{attribute 'no_explicit_call' := 'do not call this function block directly'} 
FUNCTION_BLOCK ABSTRACT GenericList EXTENDS Object IMPLEMENTS IList
VAR_INPUT
	DefaultAllocationElemetsCount : BYTE := 10;	
END_VAR
VAR_OUTPUT
	StoredTypeCategory : TYPE_CATEGORY;
END_VAR
VAR
	_Array : POINTER TO GENERIC_VALUE;
	_ArrayLength : DINT;
	_ValueCount : DINT;
END_VAR

METHOD AllocateMemory
VAR_INPUT
	elementsCount : DINT;
END_VAR
VAR	
	newMemory : POINTER TO GENERIC_VALUE;
END_VAR
newMemory := __NEW(BYTE, TO_UDINT(SIZEOF(GENERIC_VALUE) * (_ArrayLength + elementsCount)));

IF _ValueCount > 0 THEN
	Tc2_System.MEMCPY(newMemory, _Array, TO_UDINT(SIZEOF(GENERIC_VALUE) * _ValueCount));
END_IF
 
IF _Array <> 0 THEN
	__DELETE(_Array);
END_IF

_ArrayLength := _ArrayLength + elementsCount;

_Array := newMemory;
END_METHOD

METHOD Append : DINT
VAR_INPUT
	value : ANY;
	isObject : BOOL := FALSE;
END_VAR
VAR
	genericValue : GENERIC_VALUE;
END_VAR
genericValue.FromAnyType(value, isObject, StoredTypeCategory = TYPE_CATEGORY.VALUE_TYPE);

Append := AppendGenericValue(genericValue);
END_METHOD

METHOD PROTECTED AppendGenericValue : DINT
VAR_IN_OUT CONSTANT
	value : GENERIC_VALUE;
END_VAR
AppendGenericValue := _ValueCount;

InsertGenericValue(value, AppendGenericValue);
END_METHOD

METHOD Clear
VAR
	i : DINT;
END_VAR
IF _ValueCount > 0 AND_THEN StoredTypeCategory = TYPE_CATEGORY.VALUE_TYPE THEN
	FOR i := 0 TO _ValueCount - 1 DO
		_Array[i].ReleaseOwnedMemory();						
	END_FOR	
END_IF

_ValueCount := 0;
_ArrayLength := 0;

IF _Array <> 0 THEN
	__DELETE(_Array);	
END_IF
END_METHOD

{attribute 'OPC.UA.DA.Property' := '1'}
{attribute 'monitoring' := 'call'}
PROPERTY Count : DINT
GET
Count := _ValueCount;
END_GET
END_PROPERTY

METHOD CreateEnumerator : IEnumerator
VAR
	listEnumerator : POINTER TO ListEnumerator;
END_VAR
listEnumerator := __NEW(ListEnumerator(list := THIS^));

CreateEnumerator := listEnumerator^;
END_METHOD

METHOD FB_exit : BOOL
VAR_INPUT
	bInCopyCode : BOOL; // if TRUE, the exit method is called for exiting an instance that is copied afterwards (online change).
END_VAR
Clear();
END_METHOD

METHOD FindSingle : BOOL
VAR_INPUT
	predicate : IPredicate;
	skip : UDINT := 0;
	searchDirection : SEARCH_DIRECTION := SEARCH_DIRECTION.FROM_BEGINNING;
END_VAR
VAR_OUTPUT
	value : GENERIC_VALUE;
	index : DINT;
END_VAR
VAR
	startSearchIndex : DINT;
	maxSearchIndex : DINT;
	indexStep : DINT;
	i : DINT;
	skiped : UDINT := 0;
END_VAR
index := 0;
	
IF TO_DINT(skip) >= _ValueCount OR_ELSE predicate = 0 THEN
	RETURN;
END_IF

startSearchIndex := SEL(searchDirection = SEARCH_DIRECTION.FROM_BEGINNING, _ValueCount - 1, 0);
maxSearchIndex := SEL(searchDirection = SEARCH_DIRECTION.FROM_BEGINNING, 0, _ValueCount - 1);
indexStep := SEL(searchDirection = SEARCH_DIRECTION.FROM_BEGINNING, -1, 1);

FOR i := startSearchIndex TO maxSearchIndex BY indexStep DO
	IF predicate.Compare(_Array[i].AsAnyType()) THEN
		IF skip = skiped THEN
			value := _Array[i];
			index := i;
			FindSingle := TRUE;
			RETURN;
		ELSE
			skiped := skiped + 1;
		END_IF
	END_IF
END_FOR
END_METHOD

METHOD Get : REFERENCE TO GENERIC_VALUE
VAR_INPUT
	index : DINT;
END_VAR
VAR
	argumentOutOfRangeException : ArgumentOutOfRangeException;
END_VAR
IF index < 0 OR index >= _ValueCount THEN
	argumentOutOfRangeException.Throw(CurrentNamespace.Name, ClassName, __POUNAME(), __POSITION(), 'index', index);
END_IF

Get REF= _Array[index];
END_METHOD

METHOD Insert
VAR_INPUT
	value : ANY;
	index : DINT;
	isObject : BOOL := FALSE;
END_VAR
VAR
	genericValue : GENERIC_VALUE;
END_VAR
genericValue.FromAnyType(value, isObject, StoredTypeCategory = TYPE_CATEGORY.VALUE_TYPE);

InsertGenericValue(genericValue, index);
END_METHOD

METHOD PROTECTED InsertGenericValue
VAR_IN_OUT CONSTANT
	value : GENERIC_VALUE;	
END_VAR
VAR_INPUT
	index : DINT;
END_VAR
VAR
	argumentOutOfRangeException : ArgumentOutOfRangeException;
	i : DINT;
END_VAR
IF index < 0 OR index > _ValueCount THEN
	argumentOutOfRangeException.Throw(CurrentNamespace.Name, ClassName, __POUNAME(), __POSITION(), 'index', index);
END_IF

IF _ValueCount >= _ArrayLength THEN
	AllocateMemory(DefaultAllocationElemetsCount);
END_IF

_ValueCount := _ValueCount + 1;

i := _ValueCount - 1;

WHILE i > index DO
	_Array[i] := _Array[i - 1];	
	i := i - 1;
END_WHILE

_Array[i] := value;
END_METHOD

METHOD RemoveAt
VAR_INPUT
	index : DINT;
END_VAR
VAR
	argumentOutOfRangeException : ArgumentOutOfRangeException;

	i : DINT;
END_VAR
IF index < 0 OR index >= _ValueCount THEN
	argumentOutOfRangeException.Throw(CurrentNamespace.Name, ClassName, __POUNAME(), __POSITION(), 'index', index);
END_IF

IF StoredTypeCategory = TYPE_CATEGORY.VALUE_TYPE THEN
	_Array[index].ReleaseOwnedMemory();			
END_IF

FOR	i := index TO _ValueCount - 2 DO
	_Array[i] := _Array[i + 1];
END_FOR			
	
_ValueCount := _ValueCount - 1;
END_METHOD

METHOD RemoveFirst : BOOL
VAR_INPUT
	value : ANY;
	isObject : BOOL := FALSE;
END_VAR
VAR
	genericValue : GENERIC_VALUE;
END_VAR
genericValue.FromAnyType(value, isObject, FALSE);

RemoveFirst := RemoveFirstGenericValue(genericValue);
END_METHOD

METHOD PROTECTED RemoveFirstGenericValue : BOOL
VAR_IN_OUT CONSTANT
	value : GENERIC_VALUE;
END_VAR
VAR
	argumentOutOfRangeException : ArgumentOutOfRangeException;

	i : DINT;
END_VAR
IF _ValueCount > 0 THEN
	FOR i := 0 TO _ValueCount - 1 DO
		IF GenericValueHelper.CompareByData(_Array[i], value) THEN
			RemoveAt(i);
			RemoveFirstGenericValue := TRUE;
			RETURN;
		END_IF
	END_FOR
END_IF
END_METHOD

METHOD RemoveMatched : DINT
VAR_INPUT
	predicate : IPredicate;
	skip : UDINT := 0;
	maxRemoved : UDINT := 16#FFFFFFFF;
END_VAR
VAR
	i : DINT;
	skiped : UDINT := 0;
END_VAR
IF TO_DINT(skip) >= _ValueCount OR_ELSE predicate = 0 OR_ELSE maxRemoved = 0 THEN
	RETURN;
END_IF

FOR i := _ValueCount - 1 TO 0 BY -1 DO
	IF predicate.Compare(_Array[i].AsAnyType()) THEN
		IF skip <= skiped THEN
			RemoveAt(i);
			RemoveMatched := RemoveMatched + 1;
		ELSE
			skiped := skiped + 1;
		END_IF
	END_IF
END_FOR
END_METHOD

METHOD Set
VAR_INPUT
	value : ANY;
	index : DINT;
	isObject : BOOL := FALSE;
END_VAR
VAR
	genericValue : GENERIC_VALUE;
END_VAR
genericValue.FromAnyType(value, isObject, StoredTypeCategory = TYPE_CATEGORY.VALUE_TYPE);

SetGenericValue(genericValue, index);
END_METHOD

METHOD PROTECTED SetGenericValue 
VAR_IN_OUT CONSTANT
	value : GENERIC_VALUE;	
END_VAR
VAR_INPUT
	index : DINT;
END_VAR
VAR
	argumentOutOfRangeException : ArgumentOutOfRangeException;
END_VAR
IF index < 0 OR index >= _ValueCount THEN
	argumentOutOfRangeException.Throw(CurrentNamespace.Name, ClassName, __POUNAME(), __POSITION(), 'index', index);
END_IF

IF NOT GenericValueHelper.CompareByReferences(_Array[index], value) THEN
	_Array[index].ReleaseOwnedMemory();	
	_Array[index] := value;
END_IF
END_METHOD

{attribute 'monitoring' := 'call'}
PROPERTY Size : ULINT
GET
Size := XSIZEOF(THIS^);
END_GET
END_PROPERTY

METHOD Sort
VAR_INPUT
	comparer : IComparer;
	direction : SORT_DIRECTION := SORT_DIRECTION.ASCENDING;
END_VAR
VAR
	argumentNullException : ArgumentNullException;
	replaced : BOOL;
	i : DINT;
	comparisionResult : COMPARISION_RESULT;
END_VAR
IF comparer = 0 THEN
	argumentNullException.Throw(CurrentNamespace.Name, ClassName, __POUNAME(), __POSITION(), 'comparer');
END_IF

REPEAT
	replaced := FALSE;
	
	IF _ValueCount > 1 THEN
		FOR i := 0 TO _ValueCount - 2 DO
			comparisionResult := comparer.Compare(_Array[i], _Array[i + 1]);
			
			IF direction = SORT_DIRECTION.ASCENDING THEN
				IF comparisionResult = COMPARISION_RESULT.LEFT_GREATER_RIGHT THEN
					Swap(i, i + 1);
					replaced := TRUE;
				END_IF
			ELSE
				IF comparisionResult = COMPARISION_RESULT.LEFT_LESS_RIGHT THEN
					Swap(i, i + 1);
					replaced := TRUE;
				END_IF			
			END_IF
		END_FOR		
	END_IF
UNTIL
	NOT replaced
END_REPEAT
END_METHOD

METHOD Swap
VAR_INPUT
	index1 : DINT;
	index2 : DINT;
END_VAR
VAR
	argumentOutOfRangeException : ArgumentOutOfRangeException;
	tmp : GENERIC_VALUE;
END_VAR
IF index1 = index2 THEN
	RETURN;
ELSIF index1 < 0 OR_ELSE index1 >= _ValueCount THEN
	argumentOutOfRangeException.Throw(CurrentNamespace.Name, ClassName, __POUNAME(), __POSITION(), 'index1', index1);
ELSIF index2 < 0 OR_ELSE index2 >= _ValueCount THEN
	argumentOutOfRangeException.Throw(CurrentNamespace.Name, ClassName, __POUNAME(), __POSITION(), 'index2', index2);
END_IF

tmp := _Array[index1];
_Array[index1] := _Array[index2];
_Array[index2] := tmp;
END_METHOD

END_FUNCTION_BLOCK

(* stored: Version 1.1.0.1
   POU GenericList: Id {423efb90-4c6a-41e3-8889-647ff943b33e}, SpecialFunc None
   Folder Service members: Id {0d533e4f-b659-498e-bda5-8917c32d3bcb}
   Method AllocateMemory: Id {7805ad4a-1088-4228-99dd-d8b7fe4579c3}
   Method Append: Id {c48f84f5-3206-4f8e-a06b-95fdd5877efa}
   Method AppendGenericValue: Id {f1ff6a71-50a0-45d9-ae86-164a44b67bf8}
   Method Clear: Id {6eeb2dd8-b2fb-4bd3-af28-3d4655f329b4}
   Property Count: Id {8b78c4a9-2b51-4df9-a89b-35d75f4063d7}
   Get Get: Id {40434b4f-ac59-4ed2-adb0-38a6ead17ebd}
   Method CreateEnumerator: Id {9c229dd9-393b-46ff-976f-739fe26eedc5}
   Method FB_exit: Id {8d8b7b19-3218-490a-a08e-e708f6895db1}
   Method FindSingle: Id {5bd8df97-f8f3-46ed-97e0-2baa71205501}
   Method Get: Id {35156606-e33f-4fd7-a3f8-50e4c6feea06}
   Method Insert: Id {7c5e7ea9-1602-45c2-9555-47aa08559820}
   Method InsertGenericValue: Id {2dcf43ab-5d4d-40f0-ba4f-54f191c32509}
   Method RemoveAt: Id {0e28301b-e63b-49ca-a697-ef9528fc2481}
   Method RemoveFirst: Id {ab28382f-e74f-44a6-bee2-f905f3030356}
   Method RemoveFirstGenericValue: Id {fcd9bede-6419-44be-ad0a-030fdc1d5c4b}
   Method RemoveMatched: Id {e5cc38ae-8b20-4e35-acc9-fcd84e9d10bd}
   Method Set: Id {e9638d43-e88c-48cb-a07f-937c5e87c232}
   Method SetGenericValue: Id {28fb4746-7d53-4b08-a432-54d437f989bb}
   Property Size: Id {b8f1c23e-6bde-4d17-b77f-f3d1373a6f6b}
   Get Get: Id {0c60dbce-56ff-4644-ae28-c3c705772b31}
   Method Sort: Id {cd2a8a15-72bb-44f7-9e5d-ecb76fed56a8}
   Method Swap: Id {eb0e8297-edd7-472f-a573-82e2ae740339} *)
